(* CoDeSys 2.3.9.55 project: 5_hospital.pro *)
(* Libraries: Standard.lib 8.11.10 13:37:48 *)

(* PLC configuration (modules and I/O channels)
_Y1 AT %QX4.0 [BOOLOnX_Q] Ch_1 Digital output
_Y2 AT %QX4.1 [BOOLOnX_Q] Ch_2 Digital output
_Y3 AT %QX4.2 [BOOLOnX_Q] Ch_3 Digital output
_PCH1 AT %QX4.3 [BOOLOnX_Q] Ch_4 Digital output
_PCH2 AT %QX4.4 [BOOLOnX_Q] Ch_5 Digital output
_Pump AT %QX4.5 [BOOLOnX_Q] Ch_6 Digital output
_Spare1 AT %QX4.6 [BOOLOnX_Q] Ch_7 Digital output
_Spare2 AT %QX4.7 [BOOLOnX_Q] Ch_8 Digital output
_Heater AT %QW0 [WORDOnW_Q] Ch_1 Analog output
_Cooler AT %QW1 [WORDOnW_Q] Ch_2 Analog output
_Spare_AO1 AT %QW2 [WORDOnW_Q] Ch_3 Analog output
_SpareAO2 AT %QW3 [WORDOnW_Q] Ch_4 Analog output
0750-1405 16 DI 24V DC 3.0ms [Type_1_16_Channels] node 0, in %IB16 out %QB8
  _HeaterAirIn AT %IX8.0 [BOOLOnX_I] Ch_1 Digital input
  _Dust_N1 AT %IX8.1 [BOOLOnX_I] Ch_2 Digital input
  _Dust_N2 AT %IX8.2 [BOOLOnX_I] Ch_3 Digital input
  _Alm_N1 AT %IX8.3 [BOOLOnX_I] Ch_4 Digital input
  _Alm_N2 AT %IX8.4 [BOOLOnX_I] Ch_5 Digital input
  _Dust_N3 AT %IX8.5 [BOOLOnX_I] Ch_6 Digital input
  _HeatProtect_M1 AT %IX8.6 [BOOLOnX_I] Ch_7 Digital input
  _HeatProtect_M2 AT %IX8.7 [BOOLOnX_I] Ch_8 Digital input
  _DryRotationProtect AT %IX8.8 [BOOLOnX_I] Ch_9 Digital input
  _MotorProtect_M1 AT %IX8.9 [BOOLOnX_I] Ch_10 Digital input
  _RotationInv_1 AT %IX8.10 [BOOLOnX_I] Ch_11 Digital input
  _RotationInv_2 AT %IX8.11 [BOOLOnX_I] Ch_12 Digital input
  AT %IX8.12 [BOOLOnX_I] Ch_13 Digital input
  AT %IX8.13 [BOOLOnX_I] Ch_14 Digital input
  AT %IX8.14 [BOOLOnX_I] Ch_15 Digital input
  AT %IX8.15 [BOOLOnX_I] Ch_16 Digital input
_AirTemp AT %IW0 [INTOnW_I] Ch_1 signed Input value
_BackPlumpTemp AT %IW1 [INTOnW_I] Ch_2 signed Input value
_PritochTemp AT %IW2 [INTOnW_I] Ch_3 signed Input value
AT %IW3 [INTOnW_I] Ch_4 signed Input value
AT %IW4 [INTOnW_I] Ch_5 signed Input value
AT %IW5 [INTOnW_I] Ch_6 signed Input value
AT %IW6 [INTOnW_I] Ch_7 signed Input value
AT %IW7 [INTOnW_I] Ch_8 signed Input value
Fieldbus variables [FB_VARS] node 1, in %IB0 out %QB0
Flag variables [FLAG_VARS] node 2, in %IB0 out %QB0
Modbus-Master [MB_MASTER] node 3, in %IB0 out %QB0
*)

(* Global variable list: _DO *)
VAR_GLOBAL
	Y1	:	BOOL;
	Y2	:	BOOL;
	Y3	:	BOOL;
	PCH1	:	BOOL;
	PCH2	:	BOOL;
	Pump	:	BOOL;

	wDO AT %MW1000:	WORD;

END_VAR

(* Global variable list: AI *)
VAR_GLOBAL
	AirTemp	AT %MW100:	REAL;
	BackPlumpTemp	AT %MW104:	REAL;
	PritochTemp	AT %MW108:	REAL;

END_VAR

(* Global variable list: Alm *)
VAR_GLOBAL

	xResetAllAlm AT %MW200:	BOOL;
	xResetAlm_M1 AT %MW204:	BOOL;
	xResetAlm_M2 AT %MW208:	BOOL;

	wAlm_Motor_M1 AT %MW212: WORD;
	wAlm_Motor_M2 AT %MW216:	WORD;
	wAlm_WaterMotor AT %MW220:	WORD;
	wAllAlm AT %MW228:	WORD;
	xAllAlm AT %MW224:	WORD;
END_VAR

(* Global variable list: AO *)
VAR_GLOBAL

	Heater	:	WORD;
	Cooler	:	WORD;
	SpareAO1	:	WORD;
	SpareAO2	:	WORD;


END_VAR

(* Global variable list: Cooler *)
VAR_GLOBAL
	CoolerPowerSet_1 AT %MW300: REAL;
END_VAR

(* Global variable list: DI *)
VAR_GLOBAL

	HeaterAirIn	:	BOOL;
	DustN1	:	BOOL;
	DustN2	:	BOOL;
	AlmN1	:	BOOL;
	AlmN2	:	BOOL;
	DustN3	:	BOOL;
	HeatProtectM1	:	BOOL;
	HeatProtectM2	:	BOOL;
	DryRotationProtect	:	BOOL;
	MotorProtectM1	:	BOOL;
	RotationInv1	:	BOOL;
	RotationInv2	:	BOOL;
	wDI AT %MW1010:	WORD;



END_VAR

(* Global variable list: Heater *)
VAR_GLOBAL
	HeaterPowerSet_1 AT %MW400 : REAL;
	HeaterFeadBack AT %MW408 : REAL;
END_VAR

(* Global variable list: Motors *)
VAR_GLOBAL
	xVentStart:BOOL;
	xWaterMotorStart: BOOL;
	Ymotor: BOOL;

END_VAR

(* Global variable list: Process *)
VAR_GLOBAL
	wState AT %MW500	:	WORD;
	xStartProc AT %MW504: BOOL;
	xStart AT %MW508: BOOL;
	xStop AT %MW512: BOOL;
END_VAR

(* Global variable list: Settings *)
VAR_GLOBAL RETAIN

	HeaterSet_T AT %MW600 :REAL:=20;

	HeaterPowerMode AT %MW604:	BOOL;


	HeaterSet_P AT %MW608 : REAL;


	Heater_Kp AT %MW612: REAL:=10;
	Heater_Ki AT %MW616: REAL:=15;
	Heater_Kd AT %MW620: REAL;

	HeaterwMaxPower AT %MW624: WORD:=100;

	StartTemp AT %MW628: REAL:=10;

	wFroasenTemp AT %MW632:	REAL:=8;
	CoolerSet_T AT %MW636: REAL:=20;

	CoolerPowerMode AT %MW640:	BOOL;


	CoolerSet_P AT %MW644: REAL;


	Cooler_Kp AT %MW648: REAL:=0.3;
	Cooler_Ki AT %MW652: REAL:=0.5;
	Cooler_Kd AT %MW656: REAL;

	CoolerwMaxPower AT %MW660: WORD:=100;
	PreviousTemp AT %MW664: REAL:=35;

	xStartWithSecond AT %MW668: BOOL;

END_VAR

(* POU PLC_PRG, ST *)
PROGRAM PLC_PRG
VAR
	xDebug: BOOL;
	deb: WORD;
	Heater_deb: WORD;
	Cooler_deb: WORD;
	xFirstStart: BOOL:=TRUE;
END_VAR
InToVars();

IF xFirstStart THEN
	xFirstStart:=FALSE;
	xStartProc:=TRUE;
END_IF




prValue_to_AO();
IF NOT xDebug THEN
	prPreviousHeating();
	prHeater();
	prMotor();
	VarsToOut();
ELSE
	_Heater	:=	Heater_deb;
	_Spare_AO1	:=	Cooler_deb	;
END_IF
xResetAllAlm:=FALSE;
xFirstStart:=FALSE;
END_PROGRAM

(* POU InToVars, ST *)
PROGRAM InToVars
VAR
END_VAR
HeaterAirIn	:=	_HeaterAirIn	;
DustN1	:=	_Dust_N1	;
DustN2	:=	_Dust_N2	;
AlmN1	:=	_Alm_N1	;
AlmN2	:=	_Alm_N2	;
DustN3	:=	_Dust_N3	;
HeatProtectM1	:=	_HeatProtect_M1	;
HeatProtectM2	:=	_HeatProtect_M2	;
DryRotationProtect	:=	_DryRotationProtect	;
MotorProtectM1	:=	_MotorProtect_M1	;
RotationInv1	:=	_RotationInv_1	;
RotationInv2	:=	_RotationInv_2	;
			
AirTemp	:=WORD_TO_REAL(_AirTemp)/10	;
BackPlumpTemp	:=	WORD_TO_REAL(_BackPlumpTemp)/10	;
PritochTemp	:= WORD_TO_REAL(_PritochTemp)/10	;
wDI.0	:=	HeaterAirIn	;
wDI.1	:=	DustN1	;
wDI.2	:=	DustN2	;
wDI.3	:=	AlmN1	;
wDI.4	:=	AlmN2	;
wDI.5	:=	DustN3	;
wDI.6	:=	HeatProtectM1	;
wDI.7	:=	HeatProtectM2	;
wDI.8	:=	DryRotationProtect	;
wDI.9	:=	MotorProtectM1	;
wDI.10	:=	RotationInv1	;
wDI.11	:=	RotationInv2	;
END_PROGRAM

(* POU Device/AI_Conversion/prValue_to_AO, ST *)
PROGRAM prValue_to_AO
VAR
	PumpOut_1: LIN_TRAFO;
	PumpOut_2: LIN_TRAFO;
	PumpOut_3: LIN_TRAFO;
	PumpOut_4: LIN_TRAFO;

	HeaterOut_1: LIN_TRAFO;
	HeaterOut_2: LIN_TRAFO;
	HeaterOut_3: LIN_TRAFO;
	HeaterOut_4: LIN_TRAFO;

	CoolerOut_1: LIN_TRAFO;
END_VAR
(*PumpOut_1(
	IN:= PumpSpeedSet_1,
	IN_MIN:= 0,
	IN_MAX:= 50,
	OUT_MIN:= 0,
	OUT_MAX:= 32762,
	ERROR=> );
	AO_PumpSpeedSet_1:= REAL_TO_WORD(PumpOut_1.OUT);

PumpOut_2(
	IN:= PumpSpeedSet_2,
	IN_MIN:= 0,
	IN_MAX:= 50,
	OUT_MIN:= 0,
	OUT_MAX:= 32762,
	ERROR=> );
	AO_PumpSpeedSet_2:= REAL_TO_WORD(PumpOut_2.OUT);

PumpOut_3(
	IN:= PumpSpeedSet_3,
	IN_MIN:= 0,
	IN_MAX:= 50,
	OUT_MIN:= 0,
	OUT_MAX:= 32762,
	ERROR=> );
	AO_PumpSpeedSet_3:= REAL_TO_WORD(PumpOut_3.OUT);

PumpOut_4(
	IN:= PumpSpeedSet_4,
	IN_MIN:= 0,
	IN_MAX:= 50,
	OUT_MIN:= 0,
	OUT_MAX:= 32762,
	ERROR=> );
	AO_PumpSpeedSet_4:= REAL_TO_WORD(PumpOut_4.OUT);
*)

HeaterOut_1(
	IN:= HeaterPowerSet_1,
	IN_MIN:= 0,
	IN_MAX:= 100,
	OUT_MIN:= 0,
	OUT_MAX:= 32762,
	ERROR=> );
	Heater:= REAL_TO_WORD(HeaterOut_1.OUT);

CoolerOut_1(
	IN:= CoolerPowerSet_1,
	IN_MIN:= 0,
	IN_MAX:= 100,
	OUT_MIN:= 0,
	OUT_MAX:= 32762,
	ERROR=> );
	Cooler:= REAL_TO_WORD(CoolerOut_1.OUT);
(*
HeaterOut_2(
	IN:= HeaterPowerSet_2,
	IN_MIN:= 0,
	IN_MAX:= 100,
	OUT_MIN:= 0,
	OUT_MAX:= 32762,
	ERROR=> );
	AO_HeaterPowerSet_2:= REAL_TO_WORD(HeaterOut_2.OUT);


HeaterOut_3(
	IN:= HeaterPowerSet_3,
	IN_MIN:= 0,
	IN_MAX:= 100,
	OUT_MIN:= 0,
	OUT_MAX:= 32762,
	ERROR=> );
	AO_HeaterPowerSet_3:= REAL_TO_WORD(HeaterOut_3.OUT);

HeaterOut_4(
	IN:= HeaterPowerSet_4,
	IN_MIN:= 0,
	IN_MAX:= 100,
	OUT_MIN:= 0,
	OUT_MAX:= 32762,
	ERROR=> );
	AO_HeaterPowerSet_4:= REAL_TO_WORD(HeaterOut_4.OUT);
*)
END_PROGRAM

(* POU _ExtraFB/mathematical functions/LIN_TRAFO, ST *)
(* linear transformation *)
FUNCTION_BLOCK LIN_TRAFO
VAR_INPUT
	IN: REAL;				(* input value*)
	IN_MIN:REAL;			(* minimum input value *)
	IN_MAX:REAL;			(* maximum input value *)
	OUT_MIN:REAL;		(* corresponding minimum output value *)
	OUT_MAX:REAL;		(* corresponding maximum output value *)
END_VAR
VAR_OUTPUT
	OUT: REAL;			(* output value *)
	ERROR: BOOL;		(* error: IN_MIN = IN_MAX or IN out of interval *)
END_VAR

VAR
	Diff: REAL;
END_VAR
Diff := IN_MAX-IN_MIN;
ERROR := (Diff=0) OR (IN<IN_MIN) OR (IN>IN_MAX);

IF NOT ERROR THEN
	OUT := (IN-IN_MIN)/Diff * (OUT_MAX-OUT_MIN) + OUT_MIN;
END_IF
END_FUNCTION_BLOCK

(* POU prPreviousHeating, ST *)
PROGRAM prPreviousHeating
VAR
	tnPreviousHeating: TON;
	ftStart:	F_TRIG;
	rtStart:	R_TRIG;
	rtStop:	R_TRIG;
END_VAR
IF (NOT  HeaterAirIn) OR BackPlumpTemp < wFroasenTemp THEN
	wState:= 66;
END_IF
rtStart(CLK:=xStart);
IF rtStart.Q THEN
	xStartProc:=TRUE;
END_IF

rtStop(CLK:=xStop);
IF rtStop.Q THEN
	xStartProc:=FALSE;
END_IF

ftStart(CLK:=xStartProc);
IF ftStart.Q THEN
	xResetAllAlm:=TRUE;
	wState:= 0;
END_IF

CASE wState OF


			0:

				Y1:= FALSE;
				xVentStart:=FALSE;
				(*
				IF AirTemp > 19 THEN
					HeaterPowerMode:=TRUE;
					CoolerPowerMode:=TRUE;
					xWaterMotorStart:=FALSE;
					HeaterSet_P:=0;
					CoolerSet_P:=0;
				ELSE
					HeaterFeadBack:=BackPlumpTemp;
					HeaterPowerMode:=FALSE;;
					xWaterMotorStart:=TRUE;
				END_IF
*)
				HeaterFeadBack:=BackPlumpTemp;
				HeaterPowerMode:=FALSE;;
				xWaterMotorStart:=TRUE;
				IF xStartProc THEN
					wState:=1;
				END_IF



			1:

				IF AirTemp > 19 THEN
					wState:=100;
				ELSE
					wState:=10;
				END_IF


			10:

				xWaterMotorStart:=TRUE;
				HeaterPowerMode:=TRUE;
				HeaterSet_P:=100;
				CoolerPowerMode:=TRUE;
				CoolerSet_P:=0;
				IF BackPlumpTemp > StartTemp AND BackPlumpTemp < 850 THEN
					wState:=11;

				END_IF
				IF AirTemp > 19 THEN
					wState:=100;
				END_IF


			11:

				xWaterMotorStart:=TRUE;
				CoolerPowerMode:=TRUE;
				CoolerSet_P:=0;
				HeaterFeadBack:=PritochTemp;
				IF Pump THEN
					HeaterPowerMode:=FALSE;
					Y1:= TRUE;
					Ymotor:= TRUE;
					xVentStart:=TRUE;
				ELSE
					HeaterPowerMode:=TRUE;
					HeaterSet_P:=0;
					Y1:= FALSE;
					Ymotor:=FALSE;
					xVentStart:=FALSE;
				END_IF

				IF AirTemp > 19 THEN
					wState:=100;
				END_IF



			100:

				HeaterPowerMode:=TRUE;
				xWaterMotorStart:=TRUE;
				HeaterSet_P:=0;
				CoolerPowerMode:=FALSE;
				Y1:= TRUE;
				Ymotor:= TRUE;
				xVentStart:=TRUE;


			66:


				xWaterMotorStart:=TRUE;
				HeaterPowerMode:=TRUE;
				HeaterSet_P:=100;
				CoolerPowerMode:=TRUE;
				CoolerSet_P:=0;
				Y1:= FALSE;
				Y2:=FALSE;
				Y3:=FALSE;
				xVentStart:=FALSE;
				IF BackPlumpTemp > 12 AND BackPlumpTemp < 850 AND HeaterAirIn THEN
					wState:=0;
				END_IF


END_CASE
END_PROGRAM

(* POU Device/Heater/prHeater, ST *)
PROGRAM prHeater
VAR
	Heater: fbHeater;
	Cooler: fbHeater;
	wTmanualSet: REAL;
	CoolerSet: REAL;
END_VAR
Heater(
	xManualMode:= TRUE,
	xNoFeedback:= HeaterPowerMode,
	wTautoSet:=HeaterSet_T ,
	wPowerManualSet:= HeaterSet_P,
	wKp:= Heater_Kp,
	wKi:= Heater_Ki,
	wKd:= Heater_Kd,
	wMaxPower:= HeaterwMaxPower,
	wMinPower:= ,
	wTget:= (*PritochTemp*)HeaterFeadBack,
	wFlawGet:= 100,
	xInterlock:= ,
	xPumpWorking:= TRUE ,
	wTmanualSet:= HeaterSet_T,
	wAO_Power=> HeaterPowerSet_1,
	wError=> );
CoolerSet:= 50 - CoolerSet_T;
Cooler(
	xManualMode:= TRUE,
	xNoFeedback:= CoolerPowerMode,
	wTautoSet:=CoolerSet ,
	wPowerManualSet:= CoolerSet_P,
	wKp:= Cooler_Kp,
	wKi:= Cooler_Ki,
	wKd:= Heater_Kd,
	wMaxPower:= CoolerwMaxPower,
	wMinPower:= ,
	wTget:=50 - PritochTemp,
	wFlawGet:= 100,
	xInterlock:= ,
	xPumpWorking:= TRUE,
	wTmanualSet:= CoolerSet,
	wAO_Power=> CoolerPowerSet_1,
	wError=> );
END_PROGRAM

(* POU Device/Heater/fbHeater, ST *)
FUNCTION_BLOCK fbHeater
VAR_INPUT
	xManualMode:			BOOL;
	xNoFeedback:			BOOL;
	wTautoSet:			REAL;
	wPowerManualSet:	REAL;
	wKp:					REAL;
	wKi:					REAL;
	wKd:					REAL;
	wMaxPower:			WORD;
	wMinPower:			WORD;
	wTget:					REAL;
	wFlawGet:				REAL;
	xInterlock:				BOOL;
	xPumpWorking:		BOOL;
END_VAR
VAR_IN_OUT
	wTmanualSet:			REAL;
END_VAR
VAR_OUTPUT
	wAO_Power:			REAL;
	wError:					WORD;
END_VAR
VAR
	fbAutoPID:				fbPID;
	tnNoFlaw:				TON;
	rtReset:	R_TRIG;
	RESET: BOOL;
END_VAR
IF xManualMode THEN
	IF (wTmanualSet > 0 OR xNoFeedback) AND wError = 0 THEN
		rtReset(CLK:=fbAutoPID.OVERFLOW);
		IF rtReset.Q THEN
			RESET:=TRUE;
		END_IF
		fbAutoPID(
			ACTUAL:= wTget,
			SET_POINT:= wTmanualSet,
			KP:= wKp,
			TN:= wKi,
			TV:= wKd,
			Y_MANUAL:= wPowerManualSet,
			Y_OFFSET:= ,
			Y_MIN:= wMinPower,
			Y_MAX:= wMaxPower,
			MANUAL:= xNoFeedback,
			RESET:= RESET,
			Y=> ,
			LIMITS_ACTIVE=> ,
			OVERFLOW=> );
			wAO_Power:= fbAutoPID.Y;
	ELSE
		wAO_Power:=0;
	END_IF
ELSE
	wTmanualSet:=wTautoSet;
	IF wTautoSet > 0 AND wError = 0 THEN
		fbAutoPID(
			ACTUAL:= wTget,
			SET_POINT:= wTautoSet,
			KP:= wKp,
			TN:= wKi,
			TV:= wKd,
			Y_MANUAL:= ,
			Y_OFFSET:= ,
			Y_MIN:= wMinPower,
			Y_MAX:= wMaxPower,
			MANUAL:=FALSE ,
			RESET:= ,
			Y=> ,
			LIMITS_ACTIVE=> ,
			OVERFLOW=> );
			wAO_Power:= fbAutoPID.Y;
	ELSE
		wAO_Power:=0;
	END_IF
END_IF


RESET:=FALSE;
tnNoFlaw(IN:=  (NOT xPumpWorking) OR (wFlawGet = 0), PT:=T#20s, Q=>wError.0);
(*
IF tnNoFlaw.Q THEN
	wError.0:=TRUE;
END_IF
*)
END_FUNCTION_BLOCK

(* POU _ExtraFB/ControlFB/fbPID, ST *)
FUNCTION_BLOCK fbPID
VAR_INPUT
	ACTUAL :REAL;		(* actual value, process variable *)
	SET_POINT:REAL;	(* desired value, set point *)
	KP:REAL;				(* proportionality const. (P)*)
	TN:REAL;				(* reset time (I) in sec *)
	TV:REAL;				(* rate time, derivative time (D) in sec*)
	Y_MANUAL:REAL;		(* Y is set to this value as long as MANUAL=TRUE *)
	Y_OFFSET:REAL;		(* offset for manipulated variable *)
	Y_MIN:REAL;			(* minimum value for manipulated variable *)
	Y_MAX:REAL;			(* maximum value for manipulated variable *)
	MANUAL:BOOL;		(* 	TRUE: manual: Y is not influenced by controller,
								FALSE: controller determines Y *)
	RESET:BOOL;			(* reset: set Y output to Y_OFFSET and reset integral part *)
END_VAR
VAR_OUTPUT
	Y:REAL;				(* manipulated variable, set value*)
	LIMITS_ACTIVE:BOOL:=FALSE;	(* true set value would exceed limits Y_MIN, Y_MAX *)
	OVERFLOW:BOOL:=FALSE;		(* overflow in integral part *)
END_VAR
VAR
	CLOCK:TON;
	I: INTEGRAL;
	D: DERIVATIVE;
	TMDIFF: DWORD;
	ERROR: REAL;
	INIT: BOOL:=TRUE;
	Y_ADDOFFSET: REAL;
	KPcopy:REAL;
	TNcopy:REAL;
	TVcopy:REAL;
	rIntermediateVar:REAL;
END_VAR
IF TN>0 AND KP<> 0 AND (NOT OVERFLOW OR RESET OR MANUAL) THEN
	ERROR := SET_POINT-ACTUAL;								(* Regeldifferenz *)

	IF RESET OR MANUAL OR INIT OR (KP<>KPcopy OR TN<>TNcopy OR TV<>TVcopy) THEN							(* Reset oder Handbetrieb *)
		I(RESET:=TRUE);
		D(RESET:=TRUE);
		OVERFLOW:=FALSE;
		LIMITS_ACTIVE:=FALSE;
		IF RESET OR INIT THEN
			Y := Y_OFFSET;
			INIT:=FALSE;
			Y_ADDOFFSET := 0;
		ELSIF MANUAL THEN
			Y := Y_MANUAL;
			rIntermediateVar:=I.OUT/TN+D.OUT*TV;
			Y_ADDOFFSET := Y_MANUAL-(Y_OFFSET+KP*(ERROR)+rIntermediateVar);
			(*Y_ADDOFFSET := Y_MANUAL-(Y_OFFSET+KP*(ERROR)+(I.OUT/TN+D.OUT*TV));*)
		ELSE
			Y_ADDOFFSET := Y - Y_OFFSET - KP*ERROR;
		END_IF
		TMDIFF:=0;
		CLOCK(IN:=FALSE);									(* Timer neu starten *)
		CLOCK(PT:=t#1h, IN:=TRUE);

		TNcopy := TN;
		TVcopy := TV;
		KPcopy := KP;
	ELSE
		CLOCK;												(* Timer abfragen *)
		TMDIFF:=TIME_TO_DWORD(CLOCK.ET);					(* Zeitdifferenz seit letztem Aufruf *)
	END_IF;

	IF TMDIFF>0 THEN
		CLOCK(IN:=FALSE);									(* Timer neu starten *)
		CLOCK(PT:=t#1h, IN:=TRUE);

		D(IN:=ERROR, TM:=TMDIFF, RESET:=FALSE);				(* Differential abschätzen *)
		I(IN:=ERROR, TM:=TMDIFF, RESET:=FALSE);				(* Integral abschätzen *)

		OVERFLOW := I.OVERFLOW;
		IF NOT OVERFLOW THEN
			Y:=Y_OFFSET+KP*(ERROR)+(I.OUT/TN+D.OUT*TV) + Y_ADDOFFSET;
			IF Y>1E30 OR Y<-1E30 THEN						(* Overflow steht bevor, darf aber eigentlich nicht passieren *)
				OVERFLOW:=TRUE;
			END_IF;

			LIMITS_ACTIVE:=FALSE;
			IF Y_MAX>Y_MIN AND Y>Y_MAX  THEN				(* Stellwert-Obergrenze überschritten *)
				LIMITS_ACTIVE:=TRUE;
				IF KP<>0 THEN
					I(IN:=(Y_MAX-Y)*TN/KP,TM:=1000,RESET:=FALSE);		(* Integral korrigieren *)
				END_IF
				Y:=Y_MAX;
			END_IF;
			IF Y_MAX>Y_MIN AND Y<Y_MIN THEN					(* Stellwert-Untergrenze unterschritten *)
				LIMITS_ACTIVE:=TRUE;
				IF KP<>0 THEN
					I(IN:=(Y_MIN-Y)*TN/KP,TM:=1000,RESET:=FALSE);		(* Integral korrigieren *)
				END_IF
				Y:=Y_MIN;
			END_IF;
		END_IF;
	ELSE
		CLOCK(PT:=t#1h,IN:=TRUE);
	END_IF;

END_IF;
END_FUNCTION_BLOCK

(* POU _ExtraFB/mathematical functions/INTEGRAL, ST *)
(* function block to approximate the integral of IN over the time *)
FUNCTION_BLOCK INTEGRAL
VAR_INPUT
	IN:REAL;						(* input variable *)
	TM:DWORD;					(* time since last call in msec *)
	RESET:BOOL;					(* reset: OUT is set to zero and OVERFLOW to false *)
END_VAR
VAR_OUTPUT
	OUT:REAL;					(* value of the integral *)
	OVERFLOW:BOOL:=FALSE;	(* overflow *)
END_VAR
VAR
END_VAR
IF RESET THEN
	OUT:=0;
	OVERFLOW:=FALSE;
ELSIF NOT OVERFLOW  THEN
	IF 1E38 - IN*TM < OUT OR -1E38 - IN*TM > OUT THEN
		OVERFLOW:=TRUE;
	ELSE
		OUT:=OUT+IN*TM/1000;
	END_IF;
END_IF;
END_FUNCTION_BLOCK

(* POU _ExtraFB/mathematical functions/DERIVATIVE, ST *)
(* function block to approximate the derivative of a value *)
(* to calculate this, always four values are used in order to be as exact as possible *)
FUNCTION_BLOCK DERIVATIVE
VAR_INPUT
	IN:REAL;						(* input variable *)
	TM:DWORD;					(* time since last call in msec *)
	RESET:BOOL;					(* reset: set OUT to zero *)
END_VAR
VAR_OUTPUT
	OUT:REAL;					(* derivative *)
END_VAR
VAR
	X3,X2,X1:REAL;
	T2,T1:DWORD;
	INIT:BOOL:=TRUE;
END_VAR
IF INIT OR RESET THEN
	X1:=IN;
	X2:=IN;
	X3:=IN;
	OUT:=0;
	INIT:=FALSE;
ELSE
	IF TM>0 THEN
		OUT:=(3*(IN-X3)+X1-X2)/((3*T2+4*T1+3*TM))*1000;
		X3:=X2;
		X2:=X1;
		X1:=IN;
		T2:=T1;
		T1:=TM;
	END_IF;
END_IF;
END_FUNCTION_BLOCK

(* POU Device/Motor/prMotor, ST *)
	PROGRAM prMotor
VAR
	SwitchMotors: fbSwitchMotors;
	Motor1: fbMotor;
	Motor2: fbMotor;
	Y2_isOn: BOOL;
	HeatProtection: BOOL;
	MotorStart: BOOL;
	WaterMotor: fbWaterMotor;
	tnAlm: TON;

	rtTurnToTheSec: R_TRIG;
	tnAlmSecond:TON;
	xStart_M1: BOOL;
	xStart_M2: BOOL;
END_VAR
WaterMotor(
	DryRotationProtect:=  NOT DryRotationProtect,
	MotorProtectM1:= NOT MotorProtectM1,
	xStart:= xWaterMotorStart,
	DO_start=>Pump,
	wError=> );

SwitchMotors(
	xStartingMotorChoose:= xStartWithSecond,
	wAlmMotor_M1:= wAlm_Motor_M1,
	wAlmMotor_M2:= wAlm_Motor_M2,
	xStartVent:= xVentStart,
	xStartM1=>xStart_M1 ,
	xStartM2=> xStart_M2);

Motor1(
	Y1_isOn:=Y1 ,
	xFeadback:= AlmN1,
	HeatProtection:= HeatProtectM1,
	xStart:= xStart_M1,
	xZaslOpn:= Y3,
	xResetAllAlm:= xResetAllAlm,
	xResetMyAlm:=xResetAlm_M1,
	MotorStart=> PCH1,
	wError=>wAlm_Motor_M1 );

Motor2(
	Y1_isOn:=Y1 ,
	xFeadback:= AlmN2,
	HeatProtection:= HeatProtectM2,
	xStart:= xStart_M2,
	xZaslOpn:= Y2,
	xResetAllAlm:= xResetAllAlm,
	xResetMyAlm:=xResetAlm_M2,
	MotorStart=> PCH2,
	wError=>wAlm_Motor_M2 );
END_PROGRAM

(* POU Device/Motor/fbSwitchMotors, ST *)
FUNCTION_BLOCK fbSwitchMotors
VAR_INPUT
	xStartingMotorChoose: BOOL;
	wAlmMotor_M1: WORD;
	wAlmMotor_M2: WORD;
	xStartVent:	BOOL;
END_VAR
VAR_OUTPUT
	xStartM1:	BOOL;
	xStartM2:	BOOL;
END_VAR
VAR
END_VAR
IF xStartVent THEN
	xStartM1:=((NOT xStartingMotorChoose) OR wAlmMotor_M2 > 0) AND  wAlmMotor_M1 = 0;
	xStartM2:=(xStartingMotorChoose OR wAlmMotor_M1 > 0) AND  wAlmMotor_M2 = 0;
ELSE
	xStartM1:=FALSE;
	xStartM2:=FALSE;
END_IF
END_FUNCTION_BLOCK

(* POU Device/Motor/fbMotor, ST *)
FUNCTION_BLOCK fbMotor
VAR_INPUT
	Y1_isOn:	BOOL;
	xFeadback:	BOOL;

	HeatProtection:	BOOL;

END_VAR
VAR_IN_OUT
	xStart: BOOL;
	xZaslOpn:	BOOL;
	xResetAllAlm:	BOOL;
	xResetMyAlm:	BOOL;
END_VAR
VAR_OUTPUT
	MotorStart:BOOL;
	wError:WORD;
END_VAR

VAR
	tnZaslOpn: TON;
	tnFeadbackAlm: TON;
END_VAR
wError.0:= NOT Y1_isOn;

wError.1:=NOT HeatProtection;

tnFeadbackAlm(IN:= MotorStart AND (NOT xFeadback), PT:=T#30s);
IF tnFeadbackAlm.Q THEN
	wError.2:=TRUE;
END_IF

xZaslOpn:= xStart AND wError =0;

tnZaslOpn(IN:=xZaslOpn, PT:=T#20S, Q=>MotorStart);

IF xResetAllAlm OR xResetMyAlm THEN
	wError:=0;
	xResetMyAlm:=FALSE;
END_IF
END_FUNCTION_BLOCK

(* POU Device/Motor/fbWaterMotor, ST *)
FUNCTION_BLOCK fbWaterMotor
VAR_INPUT
	DryRotationProtect: BOOL;
	MotorProtectM1: BOOL;
END_VAR
VAR_IN_OUT
	xStart: BOOL;
END_VAR
VAR_OUTPUT
	DO_start:BOOL;
	wError:WORD;
END_VAR
VAR
END_VAR
IF xStart AND (NOT (DryRotationProtect OR MotorProtectM1)) THEN
	DO_start:=TRUE;
ELSE
	DO_start:=FALSE;
END_IF;
wError.0:=DryRotationProtect;
wError.1:=MotorProtectM1;
END_FUNCTION_BLOCK

(* POU VarsToOut, ST *)
PROGRAM VarsToOut
VAR
END_VAR
_Y1	:=	Y1	;
_Y2	:=	Y2	;
_Y3	:=	Y3	;
_PCH1	:=	PCH1	;
_PCH2	:=	PCH2	;
_Pump	:=	Pump	;

_Heater	:=	Heater	;
_Spare_AO1	:=	Cooler	;

wDO.0	:=	Y1	;
wDO.1	:=	Y2	;
wDO.2	:=	Y3	;
wDO.3	:=	PCH1	;
wDO.4	:=	PCH2	;
wDO.5	:=	Pump	;
END_PROGRAM
